{region '#Template'}
	{attribute 'Version' := '1.2.1.0'}
	{attribute 'Tags' := '"LCID": "1031", "Text": "AC, Aggregates, Cooler, Temperature"'}
	{attribute 'Tags' := '"LCID": "1033", "Text": "AC, Aggregates, Cooler, Temperature"'}
	{attribute 'Description' := '"LCID": "1031", "Text": "Aggregat Kühler Temperatur mit Ventil"'}
	{attribute 'Description' := '"LCID": "1033", "Text": "Aggregate cooler temperature with valve"'}
{endregion}
FUNCTION_BLOCK FB_BA_AC_ColT_02 EXTENDS FB_BA_AggregateB
VAR_INPUT
	fSpTSuA					: REAL;// Sollwert Temperatur kühlen // Setpoint temperature cooling
	fTSuA					: REAL;// Zuluft Temperatur // Supply air temperature
END_VAR
VAR_OUTPUT
	fPresentValue			: REAL;	
	bActiveSeqCtrl			: BOOL;
END_VAR
VAR_INPUT CONSTANT PERSISTENT
END_VAR
VAR_INPUT CONSTANT
	TFl						: FB_BA_SensorAnalog_IO;												
	TRt						: FB_BA_SensorAnalog_IO;			
	TSuACtrl				: FB_BA_AC_ColTSuACtrl;
	Vlv						: FB_BA_Vlv;
END_VAR
VAR		
END_VAR

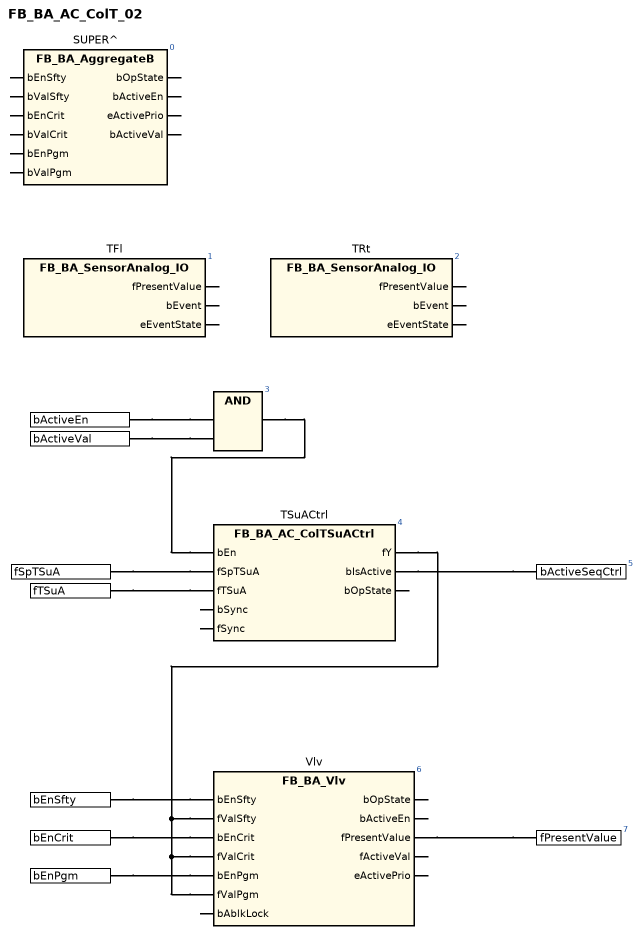
SUPER^(); // FB_BA_AggregateB
TFl(); // FB_BA_SensorAnalog_IO
TRt(); // FB_BA_SensorAnalog_IO
TSuACtrl(bEn := bActiveEn AND bActiveVal, fSpTSuA := fSpTSuA, fTSuA := fTSuA); // FB_BA_AC_ColTSuACtrl
bActiveSeqCtrl := TSuACtrl.bIsActive;
Vlv(
    bEnSfty := bEnSfty,
    fValSfty := TSuACtrl.fY,
    bEnCrit := bEnCrit,
    fValCrit := TSuACtrl.fY,
    bEnPgm := bEnPgm,
    fValPgm := TSuACtrl.fY); // FB_BA_Vlv
fPresentValue := Vlv.fPresentValue;

METHOD FB_init : BOOL
VAR_INPUT
	bInitRetains : BOOL; // if TRUE, the retain variables are initialized (warm start / cold start)
	bInCopyCode : BOOL;  // if TRUE, the instance afterwards gets moved into the copy code (online change)
END_VAR
TFl.iParent								:= THIS^;		
TFl.iLabel 								:= LblCmpAC.Cooler_TFl;	
TFl.sObjectName							:= '{Idx=41}';
TFl.eDPADMode							:= E_BA_DPADMode.eInclude;															
TFl.MV.eUnit							:= E_BA_Unit.eTemperature_DegreesCelsius;
TFl.MV.fResolution 						:= 0.01;
TFl.MV.fScaleOffset 					:= 0; 
TFl.MV.bEventDetectionEnable			:= TRUE;
TFl.MV.eEnPlantLock						:= E_BA_LockPriority.eNoLock;

TRt.iParent								:= THIS^;		
TRt.iLabel 								:= LblCmpAC.Cooler_TRt;	
TRt.sObjectName							:= '{Idx=41}';	
TRt.eDPADMode							:= E_BA_DPADMode.eInclude;																												
TRt.MV.eUnit							:= E_BA_Unit.eTemperature_DegreesCelsius;
TRt.MV.fResolution 						:= 0.01;
TRt.MV.fScaleOffset 					:= 0;  
TRt.MV.bEventDetectionEnable			:= TRUE;	
TRt.MV.eEnPlantLock						:= E_BA_LockPriority.eNoLock;

TSuACtrl.iParent						:= THIS^;	
TSuACtrl.iLabel							:= LblCmpAC.Cooler_TSuACtrl;
TSuACtrl.sObjectName					:= '{Idx=41}';										 
TSuACtrl.eDPADMode						:= E_BA_DPADMode.eInclude;								
                        				
Vlv.iParent								:= THIS^;
Vlv.iLabel								:= LblCmpAC.Cooler_Vlv;
Vlv.sObjectName							:= '{Idx=41}';										 
Vlv.eDPADMode							:= E_BA_DPADMode.eInclude;
END_METHOD

END_FUNCTION_BLOCK

(* stored: Version 1.1.0.1, ProductVersion 3.1.4024.9
   POU FB_BA_AC_ColT_02: Id {866681a9-ff68-4603-9647-0c1b945954cb}, SpecialFunc None
   Method FB_init: Id {b64f6103-0d34-457a-bb3c-2b6bc3ad8ec8} *)
